PROGRAM Aanwezigheids_lichten
VAR

END_VAR

IF GVL1.Aanwezigheidsdetector = FALSE THEN
	GVL1.Lichten := TRUE;
END_IF
IF GVL1.Aanwezigheidsdetector = TRUE THEN
	GVL1.Lichten := FALSE;
END_IF

END_PROGRAM

(* stored: Version 1.1.0.1, ProductVersion 3.1.4022.10
   POU Aanwezigheids_lichten: Id {8b76a270-81e9-4a90-9705-96adc9cad0aa}, SpecialFunc None *)
